TYPE ST_DOS_Output :
STRUCT
	bOutputCh1	: BOOL;
	bOutputCh2	: BOOL;
	bOutputCh3	: BOOL;
	bOutputCh4	: BOOL;
	bOutputCh5	: BOOL;
	bOutputCh6	: BOOL;
	bOutputCh7	: BOOL;
	bOutputCh8	: BOOL;
END_STRUCT
END_TYPE

(* stored: Version 1.1.0.1
   DUT ST_DOS_Output: Id {1520e8ca-b868-4e96-a953-15c66bdc4481} *)
